RoboDK station: kr30 cnc 090919 4.rdk

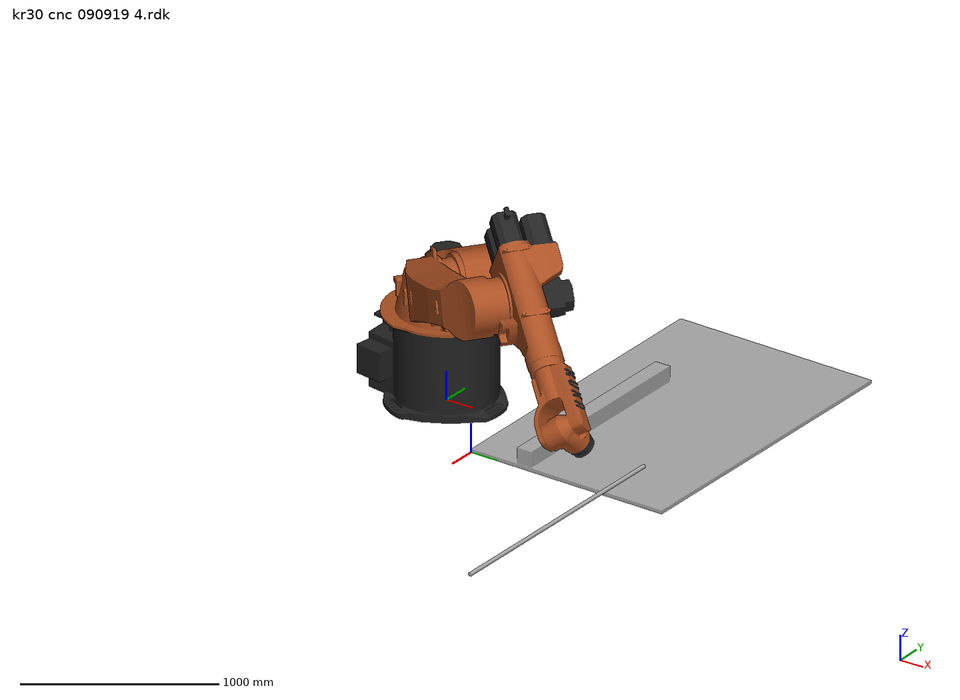
[picture v0: the station drawn from its stored meshes, robots at their saved joint values, targets as dots, program paths as lines]
Station kr30 cnc 090919 4. Poses are relative to the parent item; angles as X-Y-Z fixed-axis rotations.
  - frame KUKA KR 30 HA Base at (0, 0, 0) mm
    - robot KUKA KR 30 HA: 6 axes, payload 30 kg, reach 2033 mm, repeatability 0.05 mm, weight 665 kg
        modified DH rows (alpha deg, a mm, theta deg, d mm): 0, 0, 0, 815; -90, 350, 0, 0; 0, 850, -90, 0; -90, 145, 0, 820; 90, 0, 0, 0; -90, 0, 180, 170
        joint limits [-185, -135, -120, -350, -119, -350] to [185, 35, 158, 350, 119, 350]; home [0, -90, 90, 0, 0, 0]; saved at [36.914, -18.251, 53.387, 137.955, -69.363, -45.173]
      - tool Angle Grinder (center shaft), TCP at (165.36, 24.52, 122.34) mm, geometry from KUKA KR 30 HA
    - frame Tabletop at (921.82, -1104.91, 407.05) mm, rotated rx -0.93 ry -0.21 rz -89.9 deg
      - object kr30 tabletop mm at (-1839.9, 0, 0) mm, size 1839.9 x 1168.4 x 19 mm, geometry from kr30 tabletop mm.stl
      - object kr30 pipe jig base at (-1220, -610.6, 0) mm, size 1217.6 x 88.9 x 88.9 mm, geometry from kr30 pipe jig base.stl
      - object kr30 pipe jig pipe at (0, 0, 0) mm, size 1524 x 21.4 x 21.4 mm, geometry from kr30 pipe jig pipe.stl
